PROGRAM Bases
VAR
	
	
	
	
	IsBaseAtPlaceTrig: F_TRIG;
	IsProductLeavingTrig: F_TRIG;
	RiserFunctionality: RS;
	IsBasesClamperRiserAtLimitTrig: R_TRIG;
	TotalFinalProducts: CTU;
END_VAR

IsProductLeavingTrig(CLK:=gvl.IsProductLeaving , Q=> );
IsBaseAtPlaceTrig(CLK:=gvl.IsBaseAtPlace , Q=> );
IsBasesClamperRiserAtLimitTrig(CLK:=gvl.IsBasesClamperRiserAtLimit , Q=> );
TotalFinalProducts(
	CU:=IsProductLeavingTrig.Q , 
	RESET:=gvl.CountReset, 
	PV:= 1000, 
	Q=> , 
	CV=>gvl.ProductCounter );
CASE gvl.CurrentBaseState OF
	BaseStates.WaitingToStart:
	
	gvl.BaseConveyorMotor:=FALSE;
	gvl.BasesClamperRiserMotor:=FALSE;
	gvl.BasesClampMotor:=FALSE;

	BaseStates.LocatingBaseInPlace:
	gvl.BaseConveyorMotor:=TRUE;
	
	IF 	IsBaseAtPlaceTrig.Q THEN
		gvl.BaseConveyorMotor:=FALSE;
		gvl.BasesClampMotor:=TRUE;
		gvl.CurrentBaseState:=BaseStates.WaitingToBeLidded;
	END_IF
	
	BaseStates.Departure:
	
	RiserFunctionality(SET:=NOT gvl.IsManipulatorDectectingAnObject , RESET1:=(IsProductLeavingTrig.Q OR  gvl.IsManipulatorMovingX) , Q1=>gvl.BasesClamperRiserMotor );
	GVL.BasesClampMotor:=FALSE;
	IF  IsProductLeavingTrig.Q THEN
	Gvl.ManipulatorXMotor:=FALSE ;
	END_IF
	gvl.BaseConveyorMotor:=TRUE;
	IF IsProductLeavingTrig.Q THEN
		gvl.CurrentBaseState:=BaseStates.LocatingBaseInPlace;
	END_IF
	
	BaseStates.Stop:
	
	gvl.BaseConveyorMotor:=FALSE;
	GVL.BasesClamperRiserMotor:=FALSE;
	gvl.BasesClampMotor:=FALSE;
	
END_CASE

END_PROGRAM

(* stored: Version 1.1.0.1, ProductVersion 3.1.4024.9
   POU Bases: Id {ecc8eaa3-1bb0-4d5e-b4c7-b52ecb356e84}, SpecialFunc None *)
